PROGRAM MAIN
VAR
END_VAR

END_PROGRAM

(* stored: Version 1.1.0.1
   POU MAIN: Id {3d76308e-68d6-4f4f-af2c-a46f34e03bf0} *)
